{attribute 'GeneratedUsingTerminal: KL2300-0100'}
{attribute addProperty BoxType "KL2300-0100"}
{attribute addProperty Id "Channel_1AT %Q*Channel_70C997F30Channel_2AT %Q*Channel_70C997F30Channel_3AT %Q*Channel_70C997F30Channel_4AT %Q*Channel_70C997F30"}
{attribute addProperty CRC "3570383906"}
{attribute addProperty Size "0"}
TYPE KL_D4CFBC22 :
STRUCT
	{attribute addProperty Name "Channel_1"}
	Channel_1 : Channel_70C997F3;
	{attribute addProperty Name "Channel_2"}
	Channel_2 : Channel_70C997F3;
	{attribute addProperty Name "Channel_3"}
	Channel_3 : Channel_70C997F3;
	{attribute addProperty Name "Channel_4"}
	Channel_4 : Channel_70C997F3;
END_STRUCT
END_TYPE

(* stored: Version 1.2.0.0, ProductVersion 3.1.4024.9
   DUT KL_D4CFBC22: Id {c7dad69b-bec7-4d87-86f8-8d21ead322c3} *)
